// TIA Portal V18 export
DATA_BLOCK "shutter_DB"   // DB47
VERSION : 0.1
// stored: AutoNumber true, DBAccessibleFromOPCUA true, InstanceOfName shutter, InstanceOfType FB
"shutter"
   // VAR_INPUT
   //    "allowed OPEN" : Bool;
   //    xbh_close : Bool;
   //    xSensClosed : Bool;
   //    xSensOpen : Bool;
   //    pt_val : Time;
   // END_VAR
   // VAR_OUTPUT
   //    yPneumClose : Bool;
   //    er_no_closing : Bool;
   //    er_no_opening : Bool;
   //    er_both_activated : Bool;
   // END_VAR
   // VAR
   //    tonclos { S7_SetPoint := 'True'} : TON_TIME;
   //    tonopn { S7_SetPoint := 'True'} : TON_TIME;
   // END_VAR
   // VAR RETAIN
   //    commandClose : Bool;
   // END_VAR
   // VAR
   //    mem : Bool;
   // END_VAR
BEGIN
END_DATA_BLOCK
